// TIA Portal project "Understanding FB and FC_Training" (V16)

(* hardware
DEVICE "S71500/ET200MP station_1"  S7-1500 station
   slot 0: "Rail_0"  Rack  6ES7 590-1***0-0AA0
   slot 1: "PLC_1"  CPU 1516-3 PN/DP  6ES7 516-3AN01-0AB0  V2.8
      slot 3: "CPU display_1"  6ES7591-1BA00-0AA0
      slot 32768: "PROFINET interface_1"  X1
         slot 32769: "Port_1"  X1 P1
         slot 32770: "Port_2"  X1 P2
      slot 33024: "PROFINET interface_2"  X2
         slot 33025: "Port_1"  X2 P1
      slot 33280: "DP interface_1"  X3
      slot 34817: "Virtual CP interface port_1"  Virtual CP interface port  Virtual CP interface port
*)

// ===== PLC "PLC_1"  CPU 1516-3 PN/DP =====

VAR_GLOBAL   // PLC tag table "Default tag table"
   "b_Trigger_1" AT %M0.0 : Bool;
   "b_Trigger_2" AT %M0.1 : Bool;
   "b_DiffuseSensor_0" AT %I10.0 : Bool;
   "b_StartButton_0" AT %I10.1 : Bool;
   "b_StopButton_0" AT %I10.2 : Bool;
   "b_green_Indicator_0" AT %Q10.0 : Bool;
   "b_red_Indicator_0" AT %Q10.1 : Bool;
   "b_Trigger_3" AT %M0.2 : Bool;
   "b_Trigger_4" AT %M0.3 : Bool;
   "inputs" AT %IB10 : Byte;
   "outputs" AT %QB10 : Byte;
   "b_motor" AT %Q10.2 : Bool;
END_VAR

TYPE "ConveyorInputs"
   STRUCT
      Start : Bool;
      Stop : Bool;
      Reset : Bool;
      Sensor : Bool;
      Potentiometer : DInt;
   END_STRUCT;
END_TYPE

TYPE "ConveyorOutputs"
   STRUCT
      SpeedConveyor : DInt;
      SpeedDisplay : DInt;
      StartIndicator : Bool;
      StopIndicator : Bool;
      ResetIndicator : Bool;
   END_STRUCT;
END_TYPE

// folder: FunctionBlocks

DATA_BLOCK "conveyor_DB"   // DB2
{ S7_Optimized_Access := 'TRUE' }
VERSION : 0.1
// stored: InstanceOfName conveyor
"conveyor"
BEGIN
END_DATA_BLOCK

// folder: Functions

DATA_BLOCK "Data_block_1"   // DB1
{ S7_Optimized_Access := 'TRUE' }
VERSION : 0.1
   VAR
      count : Int;
   END_VAR
BEGIN
END_DATA_BLOCK

// folder: ParameterInstance

DATA_BLOCK "increment_1"   // DB3
{ S7_Optimized_Access := 'TRUE' }
VERSION : 0.1
// stored: InstanceOfName increment
"increment"
BEGIN
END_DATA_BLOCK

DATA_BLOCK "increment_2"   // DB4
{ S7_Optimized_Access := 'TRUE' }
VERSION : 0.1
// stored: InstanceOfName increment
"increment"
BEGIN
END_DATA_BLOCK

DATA_BLOCK "increment_3"   // DB5
{ S7_Optimized_Access := 'TRUE' }
VERSION : 0.1
// stored: InstanceOfName increment
"increment"
BEGIN
END_DATA_BLOCK

DATA_BLOCK "parameter_instance"   // DB6
{ S7_Optimized_Access := 'TRUE' }
VERSION : 0.1
   VAR
      data : Array[0..2] of DB_ANY;
      value : Int;
   END_VAR
BEGIN
END_DATA_BLOCK

// folder: (top level)

ORGANIZATION_BLOCK "Main"   // OB1, LAD, ProgramCycle
TITLE = "Main Program Sweep (Cycle)"
{ S7_Optimized_Access := 'TRUE' }
VERSION : 0.1
   VAR_INPUT
      Initial_Call : Bool;   // Initial call of this OB
      Remanence : Bool;   // =True, if remanent data are available
   END_VAR
   VAR_TEMP   // added for the SCL form of the ladder/FBD networks
      _w1 : Bool;
   END_VAR
BEGIN

REGION Network 1
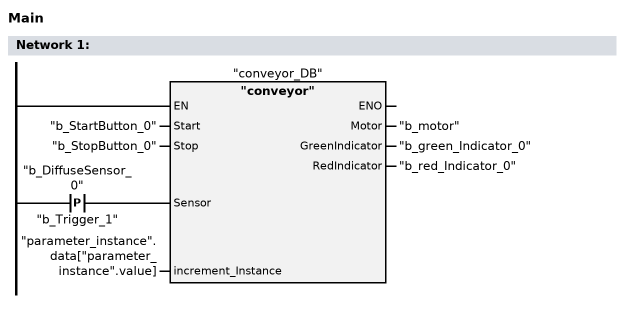
   RUNG wire#powerrail
      "conveyor_DB"(Sensor := wire#w1, Start := "b_StartButton_0", Stop := "b_StopButton_0", increment_Instance := "parameter_instance".data["parameter_instance".value], Motor => "b_motor", GreenIndicator => "b_green_Indicator_0", RedIndicator => "b_red_Indicator_0")
   END_RUNG
   RUNG wire#powerrail
      P_Contact(operand := "b_DiffuseSensor_0", bit := "b_Trigger_1")
   END_RUNG wire#w1
   // the same network as SCL:
   #_w1 := "b_DiffuseSensor_0" AND NOT "b_Trigger_1";   // rising edge of "b_DiffuseSensor_0"
   "b_Trigger_1" := "b_DiffuseSensor_0";
   "conveyor_DB"(Start := "b_StartButton_0",   // "conveyor"
                 Stop := "b_StopButton_0",
                 Sensor := #_w1,
                 increment_Instance := "parameter_instance".data["parameter_instance".value],
                 Motor => "b_motor",
                 GreenIndicator => "b_green_Indicator_0",
                 RedIndicator => "b_red_Indicator_0");
END_REGION
END_ORGANIZATION_BLOCK

ORGANIZATION_BLOCK "Startup"   // OB100, SCL, Startup
TITLE = "Complete Restart"
{ S7_Optimized_Access := 'TRUE' }
VERSION : 0.1
   VAR_INPUT
      LostRetentive : Bool;   // True if retentive data are lost
      LostRTC : Bool;   // True if date and time are lost
   END_VAR
BEGIN
   "parameter_instance".data[0] := "increment_1";
   "parameter_instance".data[1] := "increment_2";
   "parameter_instance".data[2] := "increment_3";
END_ORGANIZATION_BLOCK

// folder: FunctionBlocks

FUNCTION_BLOCK "conveyor"   // FB2, SCL
{ S7_Optimized_Access := 'TRUE' }
VERSION : 0.1
   VAR_INPUT
      Start : Bool;
      Stop : Bool;
      Sensor : Bool;
   END_VAR
   VAR_OUTPUT
      Motor : Bool;
      GreenIndicator : Bool;
      RedIndicator : Bool;
   END_VAR
   VAR_IN_OUT
      increment_Instance : "increment";
   END_VAR
   VAR
      "step" : Int;
   END_VAR
BEGIN
   IF NOT #Stop THEN
       #step := 0;
   END_IF;

   IF #Start AND #Stop THEN
       #step := 1;
   END_IF;

   IF #step = 1 THEN

       #Motor := true;
       #GreenIndicator := True;
       #RedIndicator := False;
   END_IF;

   IF #step = 0 THEN
       #Motor := false;
       #GreenIndicator := False;
       #RedIndicator := True;
   END_IF;

   #increment_Instance(In_1 := #Sensor);
END_FUNCTION_BLOCK

FUNCTION_BLOCK "decrement"   // FB3, SCL
{ S7_Optimized_Access := 'TRUE' }
VERSION : 0.1
   VAR_INPUT
      In_1 : Bool;
   END_VAR
   VAR
      count_1 : Int;
   END_VAR
BEGIN
   IF #In_1 THEN
       #count_1 := 1000 - 1;
   END_IF;
END_FUNCTION_BLOCK

// folder: Functions

FUNCTION "function_1" : Void   // FC1, SCL
{ S7_Optimized_Access := 'TRUE' }
VERSION : 0.1
   VAR_INPUT
      In_1 : Bool;
   END_VAR
   VAR_TEMP
      count : Int;
   END_VAR
BEGIN
   IF #In_1 THEN
       #count := #count + 1;
       "Data_block_1".count := "Data_block_1".count + 1;
   END_IF;
END_FUNCTION

// folder: ParameterInstance

FUNCTION_BLOCK "increment"   // FB1, SCL
{ S7_Optimized_Access := 'TRUE' }
VERSION : 0.1
   VAR_INPUT
      In_1 : Bool;
   END_VAR
   VAR
      count_2 : Int;
   END_VAR
   VAR_TEMP
      count_1 : Int;
   END_VAR
BEGIN
   IF #In_1 THEN
       #count_1 := #count_1 + 1;
       #count_2 := #count_2 + 1;
   END_IF;
END_FUNCTION_BLOCK